TYPE EspUdpEnd :
STRUCT
	EndDelimiter			: UINT := 859;
END_STRUCT
END_TYPE

(* stored: Version 1.1.0.1
   DUT EspUdpEnd: Id {1d30ec86-e764-47bf-8dc3-ba27221ffe59} *)
